TEXTLIST TextList_IAD
  0 = '' | FR: "Tension d'anode" | EN: 'Anode voltage'
  1 = '' | FR: "Courant d'anode" | EN: 'Anode current'
  2 = '' | FR: 'Courant neutraliseur' | EN: 'Neutralization current'
  3 = '' | FR: 'Pourcentage gaz 1' | EN: 'Gas 1 pourcent'
  4 = '' | FR: 'Pourcentage gaz 2' | EN: 'Gas 2 pourcent'
  5 = '' | FR: 'Durée' | EN: 'Time'
  6 = '' | FR: 'Temps écoulé' | EN: 'Elapsed time'
  7 = '' | FR: "Débit d'amorcage gaz 1" | EN: 'Starting gas 1 flow'
  8 = '' | FR: "Débit d'amorcage gaz 2" | EN: 'Starting gas 2 flow'
  9 = '' | FR: "Débit d'amorcage gaz  HCES" | EN: 'Starting gas HCES flow'
  10 = '' | FR: 'Canon à ions' | EN: 'Ions gun'
  11 = '' | FR: 'Temps' | EN: 'Time'
  12 = '' | FR: 'Temps écoulé' | EN: 'Time elapsed'
   = ''
END_TEXTLIST

(* stored: Version 1.1.0.1, ProductVersion 3.1.4024.10
   TextList TextList_IAD: Id {8e6be3c0-88bd-43cf-97ea-174e8fada12f} *)
